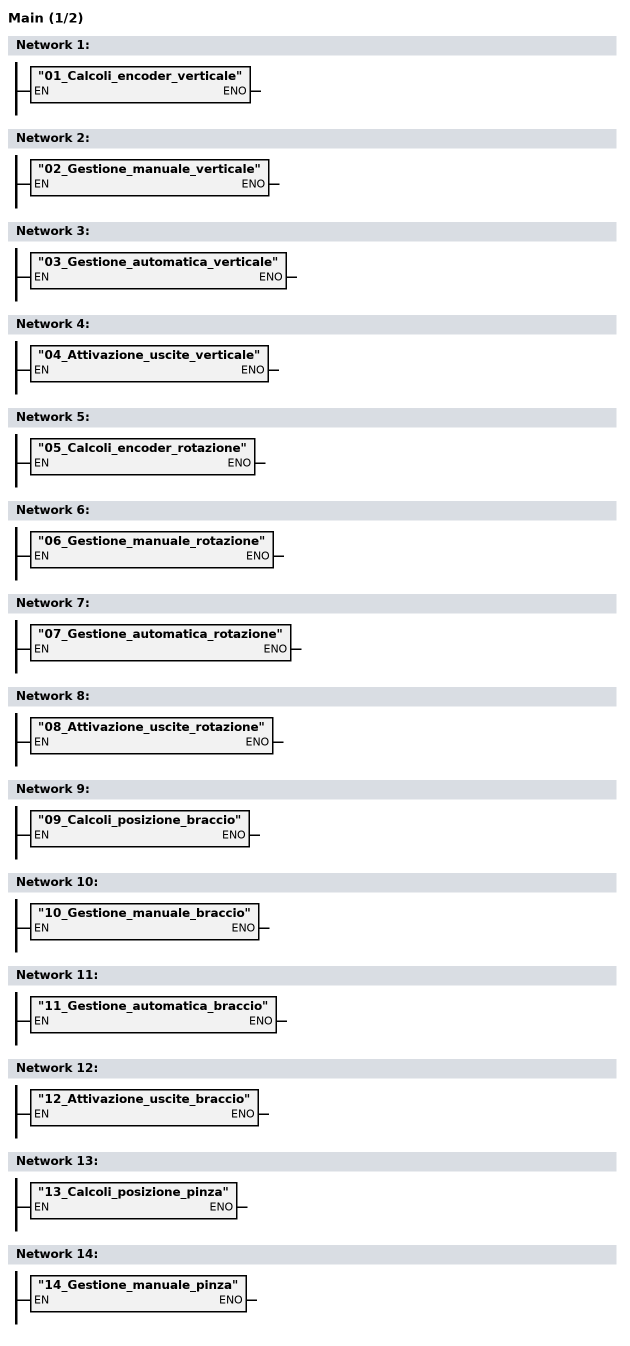
   RUNG wire#powerrail
      "01_Calcoli_encoder_verticale"()
   END_RUNG
   // the same network as SCL:
   "01_Calcoli_encoder_verticale"();
END_REGION

REGION Network 2
   RUNG wire#powerrail
      "02_Gestione_manuale_verticale"()
   END_RUNG
   // the same network as SCL:
   "02_Gestione_manuale_verticale"();
END_REGION

REGION Network 3
   RUNG wire#powerrail
      "03_Gestione_automatica_verticale"()
   END_RUNG
   // the same network as SCL:
   "03_Gestione_automatica_verticale"();
END_REGION

REGION Network 4
   RUNG wire#powerrail
      "04_Attivazione_uscite_verticale"()
   END_RUNG
   // the same network as SCL:
   "04_Attivazione_uscite_verticale"();
END_REGION

REGION Network 5
   RUNG wire#powerrail
      "05_Calcoli_encoder_rotazione"()
   END_RUNG
   // the same network as SCL:
   "05_Calcoli_encoder_rotazione"();
END_REGION

REGION Network 6
   RUNG wire#powerrail
      "06_Gestione_manuale_rotazione"()
   END_RUNG
   // the same network as SCL:
   "06_Gestione_manuale_rotazione"();
END_REGION

REGION Network 7
   RUNG wire#powerrail
      "07_Gestione_automatica_rotazione"()
   END_RUNG
   // the same network as SCL:
   "07_Gestione_automatica_rotazione"();
END_REGION

REGION Network 8
   RUNG wire#powerrail
      "08_Attivazione_uscite_rotazione"()
   END_RUNG
   // the same network as SCL:
   "08_Attivazione_uscite_rotazione"();
END_REGION

REGION Network 9
   RUNG wire#powerrail
      "09_Calcoli_posizione_braccio"()
   END_RUNG
   // the same network as SCL:
   "09_Calcoli_posizione_braccio"();
END_REGION

REGION Network 10
   RUNG wire#powerrail
      "10_Gestione_manuale_braccio"()
   END_RUNG
   // the same network as SCL:
   "10_Gestione_manuale_braccio"();
END_REGION

REGION Network 11
   RUNG wire#powerrail
      "11_Gestione_automatica_braccio"()
   END_RUNG
   // the same network as SCL:
   "11_Gestione_automatica_braccio"();
END_REGION

REGION Network 12
   RUNG wire#powerrail
      "12_Attivazione_uscite_braccio"()
   END_RUNG
   // the same network as SCL:
   "12_Attivazione_uscite_braccio"();
END_REGION

REGION Network 13
   RUNG wire#powerrail
      "13_Calcoli_posizione_pinza"()
   END_RUNG
   // the same network as SCL:
   "13_Calcoli_posizione_pinza"();
END_REGION

REGION Network 14
   RUNG wire#powerrail
      "14_Gestione_manuale_pinza"()
   END_RUNG
   // the same network as SCL:
   "14_Gestione_manuale_pinza"();
END_REGION

REGION Network 15
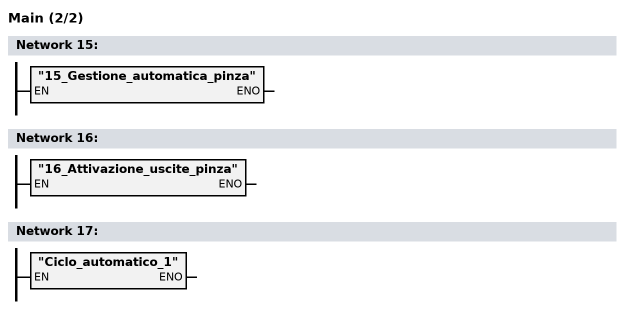
   RUNG wire#powerrail
      "15_Gestione_automatica_pinza"()
   END_RUNG
   // the same network as SCL:
   "15_Gestione_automatica_pinza"();
END_REGION

REGION Network 16
   RUNG wire#powerrail
      "16_Attivazione_uscite_pinza"()
   END_RUNG
   // the same network as SCL:
   "16_Attivazione_uscite_pinza"();
END_REGION

REGION Network 17
   RUNG wire#powerrail
      "Ciclo_automatico_1"()
   END_RUNG
   // the same network as SCL:
   "Ciclo_automatico_1"();
END_REGION
END_ORGANIZATION_BLOCK

(* ===== HMI "HMI_RT_1" =====
system functions are stored by id; their names below are inferred from use
connection "HMI_Collegamento_1": ETHERNET, SMART_S7_1200_OMS

HMI tags "Tabella delle variabili standard"
   "Variabile_Numero di pagina" : UInt, internal
   "Blocco_dati_HMI_jog_back_to_home" : Bool = PLC Blocco_dati_HMI_verticale.jog_back_to_home, 100 ms
   "Blocco_dati_HMI_jog_discesa_braccio" : Bool = PLC Blocco_dati_HMI_verticale.jog_discesa_braccio, 100 ms
   "Blocco_dati_HMI_jog_salita_braccio" : Bool = PLC Blocco_dati_HMI_verticale.jog_salita_braccio, 100 ms
   "Blocco_dati_HMI_jog_emergenza" : Bool = PLC Blocco_dati_HMI_verticale.jog_emergenza, 100 ms
   "Blocco_dati_HMI_jog_selettore_man_aut" : Bool = PLC Blocco_dati_HMI_verticale.jog_selettore_man_aut, 100 ms
   "Blocco_dati_HMI_setpoint_1" : DInt = PLC Blocco_dati_HMI_verticale.setpoint_1, 100 ms
   "Blocco_dati_HMI_setpoint_2" : DInt = PLC Blocco_dati_HMI_verticale.setpoint_2, 100 ms
   "Blocco_dati_encoder_setpoint" : DInt = PLC Blocco_dati_encoder_verticale."setpoint verticale", 100 ms
   "Blocco_dati_HMI_setpoint_3" : DInt = PLC Blocco_dati_HMI_verticale.setpoint_3, 100 ms
   "Blocco_dati_encoder_posizione vericale in mm" : DInt = PLC Blocco_dati_encoder_verticale."posizione vericale in mm", 100 ms
   "Blocco_dati_HMI_rotazione_jog_rotazione_oraria" : Bool = PLC Blocco_dati_HMI_rotazione.jog_rotazione_oraria, 100 ms
   "Blocco_dati_HMI_rotazione_jog_rotazione_antioraia" : Bool = PLC Blocco_dati_HMI_rotazione.jog_rotazione_antioraia, 100 ms
   "Blocco_dati_HMI_rotazione_jog_back_to_home_rotazione" : Bool = PLC Blocco_dati_HMI_rotazione.jog_back_to_home_rotazione, 100 ms
   "Blocco_dati_encoder_rotazione_posizione rotazione in gradi" : DInt = PLC Blocco_dati_encoder_rotazione."posizione rotazione in gradi", 100 ms
   "Blocco_dati_HMI_rotazione_setpoint_1" : DInt = PLC Blocco_dati_HMI_rotazione.setpoint_1, 100 ms
   "Blocco_dati_HMI_rotazione_setpoint_2" : DInt = PLC Blocco_dati_HMI_rotazione.setpoint_2, 100 ms
   "Blocco_dati_HMI_rotazione_setpoint_3" : DInt = PLC Blocco_dati_HMI_rotazione.setpoint_3, 100 ms
   "Blocco_dati_encoder_rotazione_setpoint rotazione" : DInt = PLC Blocco_dati_encoder_rotazione."setpoint rotazione", 100 ms
   "Blocco_dati_HMI_rotazione_jog_posizionamento_automatico_rot" : Bool = PLC Blocco_dati_HMI_rotazione.jog_posizionamento_automatico_rot, 100 ms
   "Blocco_dati_HMI_braccio_jog_avanti_braccio" : Bool = PLC Blocco_dati_HMI_braccio.jog_avanti_braccio, 1 s
   "Blocco_dati_HMI_braccio_jog_indietro_braccio" : Bool = PLC Blocco_dati_HMI_braccio.jog_indietro_braccio, 1 s
   "Blocco_dati_HMI_braccio_jog_back_to_home_orizzontale" : Bool = PLC Blocco_dati_HMI_braccio.jog_back_to_home_orizzontale, 1 s
   "Blocco_dati_contaimpulsi_braccio_posizione orizzontale in mm" : DInt = PLC Blocco_dati_contaimpulsi_braccio."posizione orizzontale in mm", 1 s
   "Blocco_dati_HMI_pinza_jog_chiusura_pinza" : Bool = PLC Blocco_dati_HMI_pinza.jog_chiusura_pinza, 1 s
   "Blocco_dati_HMI_pinza_jog_apertura_pinza" : Bool = PLC Blocco_dati_HMI_pinza.jog_apertura_pinza, 1 s
   "Blocco_dati_HMI_pinza_jog_back_to_home_pinza" : Bool = PLC Blocco_dati_HMI_pinza.jog_back_to_home_pinza, 1 s
   "Blocco_dati_HMI_braccio_setpoint_1" : DInt = PLC Blocco_dati_HMI_braccio.setpoint_1, 1 s
   "Blocco_dati_HMI_braccio_setpoint_3" : DInt = PLC Blocco_dati_HMI_braccio.setpoint_3, 1 s
   "Blocco_dati_contaimpulsi_braccio_setpoint orizzontale" : DInt = PLC Blocco_dati_contaimpulsi_braccio."setpoint orizzontale", 1 s
   "Blocco_dati_HMI_pinza_impostazione_setpoint" : DInt = PLC Blocco_dati_HMI_pinza.setpoint_1, 1 s
   "Blocco_dati_contaimpulsi_pinza_setpoint chiusura pinza" : DInt = PLC Blocco_dati_contaimpulsi_pinza."setpoint chiusura pinza", 1 s
   "conteggio impulsi pinza" : DInt = PLC "conteggio impulsi pinza" AT %MD11, 1 s
   "Blocco_dati_HMI_automatico_jog_start_automatico" : Bool = PLC Blocco_dati_HMI_automatico.jog_start_automatico, 1 s
   "Blocco_dati_HMI_verticale_setpoint_4" : DInt = PLC Blocco_dati_HMI_verticale.setpoint_4, 1 s
   "Blocco_dati_HMI_automatico_jog_ripristino" : Bool = PLC Blocco_dati_HMI_automatico.jog_ripristino, 1 s
   "Blocco_dati_HMI_pinza_setpoint_2" : DInt = PLC Blocco_dati_HMI_pinza.setpoint_2, 1 s

text list "Elenco testi_Nome della pagina": 1 'Pagina base'

Template "Modello_1" 800x480
   Button "Esci" at 714,429 size 71x50; TextOff 'Esci'; PictureOff "ExitRuntime_KTP700_Basic_PN_TR"; PictureOn "ExitRuntime_KTP700_Basic_PN_TR"
      on Release: StopRuntime(0)
   Button "Template_Button" at 614,429 size 71x50; TextOff 'Text'
   Button "Template_Button_1" at 514,429 size 71x50; TextOff 'Text'
   Button "Template_Button_2" at 414,429 size 71x50; TextOff 'Text'
   Button "Template_Button_3" at 314,429 size 71x50; TextOff 'Text'
   Button "Template_Button_4" at 214,429 size 71x50; TextOff 'Text'
   Button "Template_Button_5" at 114,429 size 71x50; TextOff 'Text'
   Button "Pagina iniziale" at 14,429 size 71x50; TextOff 'Pagina iniziale'; PictureOff "NavigateHome_KTP700_Basic_PN_TR"; PictureOn "NavigateHome_KTP700_Basic_PN_TR"
      on Release: ActivateScreen("Pagina base", 0)
   SymbolicIOField "Pagina_campo_IO_simbolico" at 93,9 size 600x33; TextOff '0'; TextOn '1'; TextList "Elenco testi_Nome della pagina"
      ProcessValue <- "Variabile_Numero di pagina"
      on Change: ActivateScreenByNumber("Variabile_Numero di pagina", 0)
   DateTimeField "HmiScreenItemData" at 695,25 size 105x25
   DateTimeField "HmiScreenItemData_1" at 695,0 size 105x25
   GraphicView "Logo" at 0,0 size 91x51; Picture "Logo di HMI_1"

screen "Pagina base" 800x480, template "Modello_1"
   on GenerateScreen: SetTag("Variabile_Numero di pagina", 1)
   TextField "HmiScreenItemData" at 80,225 size 640x25; Text 'Benvenuto in HMI_1 (KTP700 Basic+ PN)!'
   Softkey "Softkey_F1" at 0,0 size 0x0
      on KeyDown: ActivateScreen("Pagina base", 0)
   Softkey "Softkey_F2" at 0,0 size 0x0
      on KeyDown: ActivateScreen("Comandi manuali", 0)
   Softkey "Softkey_F3" at 0,0 size 0x0
      on KeyDown: ActivateScreen("Comandi automatici", 0)

screen "Comandi manuali" 800x480
   Softkey "Softkey_F1" at 0,0 size 0x0
      on KeyDown: ActivateScreen("Pagina base", 0)
   Softkey "Softkey_F2" at 0,0 size 0x0
      on KeyDown: ActivateScreen("Comandi manuali", 0)
   Softkey "Softkey_F3" at 0,0 size 0x0
      on KeyDown: ActivateScreen("Comandi automatici", 0)
   TextField "Casella di testo_1" at 319,98 size 76x20; Text 'Emergenza'
   TextField "Casella di testo_2" at 433,98 size 68x20; Text 'Man /Aut'
   TextField "Casella di testo_4" at 66,186 size 41x20; Text 'Salita'
   TextField "Casella di testo_5" at 62,384 size 65x20; Text 'Posizione'
   TextField "Casella di testo_6" at 66,323 size 35x20; Text 'Back'
   TextField "Casella di testo_7" at 66,256 size 54x20; Text 'Discesa'
   Switch "Pushbutton_Emergency" at 322,49 size 49x47; CaptionText 'Switch'; TextOff '0'; TextOn '1'; PictureOff "Pushbutton_Emergency_Off_256c"; PictureOn "Pushbutton_Emergency_On_256c"
      on SwitchOn: SetBit("Blocco_dati_HMI_jog_emergenza")
      on SwitchOff: ResetBit("Blocco_dati_HMI_jog_emergenza")
      ProcessValue <- "Blocco_dati_HMI_jog_emergenza"
   Switch "Rotary_RG" at 433,50 size 46x46; CaptionText 'Switch'; TextOff '0'; TextOn '1'; PictureOff "Rotary_RG_Off_256c"; PictureOn "Rotary_RG_On_256c"
      on SwitchOn: SetBit("Blocco_dati_HMI_jog_selettore_man_aut")
      on SwitchOff: ResetBit("Blocco_dati_HMI_jog_selettore_man_aut")
      ProcessValue <- "Blocco_dati_HMI_jog_selettore_man_aut"
   Button "FB_Up_Round" at 127,184 size 37x38; TextOff 'Text'; PictureOn "FB_Up_Round_Pressed_256c"; PictureOff "FB_Up_Round_Released_256c"
      on Press: SetBit("Blocco_dati_HMI_jog_salita_braccio")
      on Release: ResetBit("Blocco_dati_HMI_jog_salita_braccio")
   Button "FB_Down_Round" at 127,250 size 37x38; TextOff 'Text'; PictureOn "FB_Down_Round_Pressed_256c"; PictureOff "FB_Down_Round_Released_256c"
      on Press: SetBit("Blocco_dati_HMI_jog_discesa_braccio")
      on Release: ResetBit("Blocco_dati_HMI_jog_discesa_braccio")
   Button "FB_Home_Round" at 127,325 size 37x38; TextOff 'Text'; PictureOn "FB_Home_Round_Pressed_256c"; PictureOff "FB_Home_Round_Released_256c"
      on Press: SetBit("Blocco_dati_HMI_jog_back_to_home")
      on Release: ResetBit("Blocco_dati_HMI_jog_back_to_home")
   IOField "Campo I/O_1" at 314,383 size 54x29; FormatPattern 9999
      ProcessValue <- "Blocco_dati_encoder_rotazione_posizione rotazione in gradi"
   TextField "Casella di testo_10" at 62,339 size 58x20; Text 'to home'
   TextField "Casella di testo_13" at 254,188 size 45x20; Text 'Oraria'
   TextField "Casella di testo_26" at 254,325 size 35x20; Text 'Back'
   TextField "Casella di testo_27" at 244,256 size 71x20; Text 'Antioraria'
   TextField "Casella di testo_28" at 250,341 size 58x20; Text 'to home'
   IOField "Campo I/O_2" at 127,381 size 54x29; FormatPattern 9999
      ProcessValue <- "Blocco_dati_encoder_posizione vericale in mm"
   TextField "Casella di testo_3" at 247,386 size 65x20; Text 'Posizione'
   Button "FB_ArrowRight_Round" at 315,181 size 37x38; TextOff 'Text'; PictureOn "FB_ArrowRight_Round_Pressed_256c"; PictureOff "FB_ArrowRight_Round_Released_256c"
      on Press: SetBit("Blocco_dati_HMI_rotazione_jog_rotazione_oraria")
      on Release: ResetBit("Blocco_dati_HMI_rotazione_jog_rotazione_oraria")
   Button "FB_ArrowLeft_Round" at 316,250 size 36x35; TextOff 'Text'; PictureOn "FB_ArrowLeft_Round_Pressed_256c"; PictureOff "FB_ArrowLeft_Round_Released_256c"
      on Press: SetBit("Blocco_dati_HMI_rotazione_jog_rotazione_antioraia")
      on Release: ResetBit("Blocco_dati_HMI_rotazione_jog_rotazione_antioraia")
   Button "FB_Home_Round_2" at 316,326 size 36x37; TextOff 'Text'; PictureOn "FB_Home_Round_Pressed_256c"; PictureOff "FB_Home_Round_Released_256c"
      on Press: SetBit("Blocco_dati_HMI_rotazione_jog_back_to_home_rotazione")
      on Release: ResetBit("Blocco_dati_HMI_rotazione_jog_back_to_home_rotazione")
   IOField "Campo I/O_3" at 490,383 size 54x29; FormatPattern 9999
      ProcessValue <- "Blocco_dati_contaimpulsi_braccio_posizione orizzontale in mm"
   TextField "Casella di testo_15" at 430,188 size 48x20; Text 'Avanti'
   TextField "Casella di testo_16" at 430,325 size 35x20; Text 'Back'
   TextField "Casella di testo_17" at 420,256 size 57x20; Text 'Indietro'
   TextField "Casella di testo_18" at 426,341 size 58x20; Text 'to home'
   TextField "Casella di testo_19" at 423,386 size 65x20; Text 'Posizione'
   Button "FB_ArrowRight_Round_1" at 491,181 size 37x38; TextOff 'Text'; PictureOff "FB_ArrowRight_Round_Released_256c"; PictureOn "FB_ArrowRight_Round_Pressed_256c"
      on Release: ResetBit("Blocco_dati_HMI_braccio_jog_avanti_braccio")
      on Press: SetBit("Blocco_dati_HMI_braccio_jog_avanti_braccio")
   Button "FB_ArrowLeft_Round_1" at 492,250 size 36x35; TextOff 'Text'; PictureOff "FB_ArrowLeft_Round_Released_256c"; PictureOn "FB_ArrowLeft_Round_Pressed_256c"
      on Release: ResetBit("Blocco_dati_HMI_braccio_jog_indietro_braccio")
      on Press: SetBit("Blocco_dati_HMI_braccio_jog_indietro_braccio")
   Button "FB_Home_Round_1" at 492,326 size 36x37; TextOff 'Text'; PictureOff "FB_Home_Round_Released_256c"; PictureOn "FB_Home_Round_Pressed_256c"
      on Release: ResetBit("Blocco_dati_HMI_braccio_jog_back_to_home_orizzontale")
      on Press: SetBit("Blocco_dati_HMI_braccio_jog_back_to_home_orizzontale")
   IOField "Campo I/O_4" at 673,383 size 54x29; FormatPattern 9999
      ProcessValue <- "conteggio impulsi pinza"
   TextField "Casella di testo_20" at 606,188 size 61x20; Text 'Chiusura'
   TextField "Casella di testo_21" at 613,325 size 35x20; Text 'Back'
   TextField "Casella di testo_22" at 603,256 size 65x20; Text 'Apertura'
   TextField "Casella di testo_23" at 609,341 size 58x20; Text 'to home'
   TextField "Casella di testo_24" at 606,386 size 65x20; Text 'Posizione'
   Button "FB_ArrowRight_Round_2" at 674,181 size 37x38; TextOff 'Text'; PictureOn "FB_ArrowRight_Round_Pressed_256c"; PictureOff "FB_ArrowRight_Round_Released_256c"
      on Release: ResetBit("Blocco_dati_HMI_pinza_jog_chiusura_pinza")
      on Press: SetBit("Blocco_dati_HMI_pinza_jog_chiusura_pinza")
   Button "FB_ArrowLeft_Round_2" at 675,250 size 36x35; TextOff 'Text'; PictureOn "FB_ArrowLeft_Round_Pressed_256c"; PictureOff "FB_ArrowLeft_Round_Released_256c"
      on Release: ResetBit("Blocco_dati_HMI_pinza_jog_apertura_pinza")
      on Press: SetBit("Blocco_dati_HMI_pinza_jog_apertura_pinza")
   Button "FB_Home_Round_3" at 675,326 size 36x37; TextOff 'Text'; PictureOn "FB_Home_Round_Pressed_256c"; PictureOff "FB_Home_Round_Released_256c"
      on Release: ResetBit("Blocco_dati_HMI_pinza_jog_back_to_home_pinza")
      on Press: SetBit("Blocco_dati_HMI_pinza_jog_back_to_home_pinza")
   TextField "Casella di testo_9" at 303,0 size 217x29; Text 'COMANDI MANUALI'
   TextField "Casella di testo_8" at 58,138 size 145x23; Text 'ASSE VERTICALE'
   TextField "Casella di testo_11" at 250,139 size 103x23; Text 'ROTAZIONE'
   TextField "Casella di testo_12" at 455,138 size 81x23; Text 'BRACCIO'
   TextField "Casella di testo_14" at 638,138 size 57x23; Text 'PINZA'

screen "Comandi automatici" 800x480
   TextField "Casella di testo_9" at 293,8 size 222x29; Text 'CICLO AUTOMATICO'
   TextField "Casella di testo_14" at -3628,245 size 16x23; Text 'Text'
   TextField "Casella di testo_5" at 455,147 size 81x23; Text 'BRACCIO'
   TextField "Casella di testo_1" at 30,147 size 145x23; Text 'ASSE VERTICALE'
   TextField "Casella di testo_2" at 242,148 size 103x23; Text 'ROTAZIONE'
   TextField "Casella di testo_24" at 659,147 size 57x23; Text 'PINZA'
   Button "FB_Home_Round" at 524,51 size 46x45; TextOff 'Text'; PictureOn "FB_Home_Round_Pressed_256c"; PictureOff "FB_Home_Round_Released_256c"
      on Press: SetBit("Blocco_dati_HMI_automatico_jog_ripristino")
      on Release: ResetBit("Blocco_dati_HMI_automatico_jog_ripristino")
   TextField "Casella di testo_3" at 120,312 size 65x20; Text 'Posizione'
   IOField "Campo I/O_1" at 125,335 size 58x35; FormatPattern 9999
      ProcessValue <- "Blocco_dati_encoder_posizione vericale in mm"
   TextField "Casella di testo_4" at 22,194 size 67x17; Text 'Setpoint_1'
   TextField "Casella di testo_6" at 28,258 size 67x17; Text 'Setpoint_2'
   TextField "Casella di testo_7" at 26,313 size 67x17; Text 'Setpoint_3'
   TextField "Casella di testo_10" at 121,238 size 53x17; Text 'Setpoint'
   IOField "Campo I/O_3" at 38,213 size 56x25; FormatPattern 9999
      ProcessValue <- "Blocco_dati_HMI_setpoint_1"
   IOField "Campo I/O_4" at 35,279 size 56x26; FormatPattern 9999
      ProcessValue <- "Blocco_dati_HMI_setpoint_2"
   IOField "Campo I/O_5" at 35,333 size 56x26; FormatPattern 9999
      ProcessValue <- "Blocco_dati_HMI_setpoint_3"
   IOField "Campo I/O_6" at 124,259 size 55x28; FormatPattern 9999
      ProcessValue <- "Blocco_dati_encoder_setpoint"
   Button "FB_Right_Round" at 428,50 size 47x46; TextOff 'Text'; PictureOn "FB_Right_Round_Pressed_256c"; PictureOff "FB_Right_Round_Released_256c"
      on Press: SetBit("Blocco_dati_HMI_automatico_jog_start_automatico")
      on Release: ResetBit("Blocco_dati_HMI_automatico_jog_start_automatico")
   TextField "Casella di testo_8" at 221,99 size 76x20; Text 'Emergenza'
   TextField "Casella di testo_15" at 326,99 size 68x20; Text 'Man /Aut'
   Switch "Pushbutton_Emergency_1" at 224,50 size 49x47; CaptionText 'Switch'; TextOff '0'; TextOn '1'; PictureOff "Pushbutton_Emergency_Off_256c"; PictureOn "Pushbutton_Emergency_On_256c"
      on SwitchOff: ResetBit("Blocco_dati_HMI_jog_emergenza")
      on SwitchOn: SetBit("Blocco_dati_HMI_jog_emergenza")
   Switch "Rotary_RG_1" at 335,51 size 46x46; CaptionText 'Switch'; TextOff '0'; TextOn '1'; PictureOff "Rotary_RG_Off_256c"; PictureOn "Rotary_RG_On_256c"
      on SwitchOff: ResetBit("Blocco_dati_HMI_jog_selettore_man_aut")
      on SwitchOn: SetBit("Blocco_dati_HMI_jog_selettore_man_aut")
   TextField "Casella di testo_16" at 326,314 size 65x20; Text 'Posizione'
   IOField "Campo I/O_2" at 326,338 size 60x32; FormatPattern 9999
      ProcessValue <- "Blocco_dati_encoder_rotazione_posizione rotazione in gradi"
   TextField "Casella di testo_17" at 221,194 size 67x17; Text 'Setpoint_1'
   TextField "Casella di testo_18" at 221,275 size 67x17; Text 'Setpoint_2'
   TextField "Casella di testo_19" at 226,359 size 67x17; Text 'Setpoint_3'
   IOField "Campo I/O_7" at 232,211 size 56x27; FormatPattern 9999
      ProcessValue <- "Blocco_dati_HMI_rotazione_setpoint_1"
   IOField "Campo I/O_8" at 232,294 size 56x28; FormatPattern 9999
      ProcessValue <- "Blocco_dati_HMI_rotazione_setpoint_2"
   IOField "Campo I/O_9" at 235,378 size 56x28; FormatPattern 9999
      ProcessValue <- "Blocco_dati_HMI_rotazione_setpoint_3"
   IOField "Campo I/O_10" at 327,262 size 57x26; FormatPattern 9999
      ProcessValue <- "Blocco_dati_encoder_rotazione_setpoint rotazione"
   TextField "Casella di testo_20" at 325,241 size 53x17; Text 'Setpoint'
   TextField "Casella di testo_25" at 525,317 size 65x20; Text 'Posizione'
   IOField "Campo I/O_11" at 524,340 size 61x30; FormatPattern 9999
      ProcessValue <- "Blocco_dati_contaimpulsi_braccio_posizione orizzontale in mm"
   TextField "Casella di testo_26" at 420,192 size 67x17; Text 'Setpoint_1'
   TextField "Casella di testo_27" at 420,272 size 67x17; Text 'Setpoint_2'
   TextField "Casella di testo_28" at 426,359 size 67x17; Text 'Setpoint_3'
   IOField "Campo I/O_12" at 426,213 size 52x29; FormatPattern 9999
      ProcessValue <- "Blocco_dati_HMI_braccio_setpoint_1"
   IOField "Campo I/O_13" at 426,296 size 52x30; FormatPattern 9999
   IOField "Campo I/O_14" at 429,380 size 52x30; FormatPattern 9999
      ProcessValue <- "Blocco_dati_HMI_braccio_setpoint_3"
   IOField "Campo I/O_15" at 528,260 size 57x27; FormatPattern 9999
      ProcessValue <- "Blocco_dati_contaimpulsi_braccio_setpoint orizzontale"
   TextField "Casella di testo_32" at 526,239 size 53x17; Text 'Setpoint'
   TextField "Casella di testo_33" at 723,318 size 65x20; Text 'Posizione'
   IOField "Campo I/O_16" at 723,341 size 60x29; FormatPattern 9999
   TextField "Casella di testo_34" at 621,192 size 67x17; Text 'Setpoint_1'
   IOField "Campo I/O_17" at 626,215 size 57x29; FormatPattern 9999
      ProcessValue <- "Blocco_dati_HMI_pinza_impostazione_setpoint"
   IOField "Campo I/O_20" at 723,256 size 57x29; FormatPattern 9999
      ProcessValue <- "Blocco_dati_contaimpulsi_pinza_setpoint chiusura pinza"
   TextField "Casella di testo_40" at 722,231 size 53x17; Text 'Setpoint'
   TextField "Casella di testo_35" at 431,97 size 39x20; Text 'Start'
   TextField "Casella di testo_11" at 30,376 size 67x17; Text 'Setpoint_4'
   IOField "Campo I/O_18" at 34,395 size 56x26; FormatPattern 9999
      ProcessValue <- "Blocco_dati_HMI_verticale_setpoint_4"
   TextField "Casella di testo_12" at 519,95 size 66x20; Text 'Ripristino'
   IOField "Campo I/O_19" at 626,293 size 57x29; FormatPattern 9999
      ProcessValue <- "Blocco_dati_HMI_pinza_setpoint_2"
   TextField "Casella di testo_13" at 621,270 size 67x17; Text 'Setpoint_2'
   Softkey "Softkey_F3" at 0,0 size 0x0
      on KeyDown: ActivateScreen("Comandi automatici", 0)
   Softkey "Softkey_F2" at 0,0 size 0x0
      on KeyDown: ActivateScreen("Comandi manuali", 0)
   Softkey "Softkey_F1" at 0,0 size 0x0
      on KeyDown: ActivateScreen("Pagina base", 0)
*)